# EPICS substitutions: Epics_Installation/gpib_test/gpib_test/gpibApp/Db/user.substitutions
file "db/keithleyHHL.db" {
    { user = "pi" }
}
